TYPE ST_Channel :
	STRUCT
		OverVoltage : BIT ; //
		UnderVoltage : BIT ; //
		OverCurrent : BIT ; //
		PhaseSeqCW : BIT ; //
		PhaseSeqCCW : BIT ; //
		MissingZeroCrossing : BIT ; //
		TxPdoState : BIT ; //
		TxPdoToggle : BIT ; //
	END_STRUCT
END_TYPE

(* stored: Version 1.1.0.1, ProductVersion 3.1.4024.12
   DUT ST_Channel: Id {f37f7254-6ee2-47ce-9171-f9e41e1ddccf} *)
